Staubli VAL3: sendJState.pgx

public program sendJState()
  local num l_nRetVal
begin
  call sendData(siTcpIpFbk,rosJointMsg.prefix.nData,nOutConnFlag)
  call sendData(siTcpIpFbk,rosJointMsg.header.nData,nOutConnFlag)
  call sendData(siTcpIpFbk,rosJointMsg.body.nData,nOutConnFlag)
end
